Staubli VAL3: testDonneCall.pgx

program testDonneCall()
begin
  putln(sEcran,nNbPieceArrive)
end
